(*~
		<docu>
			<summary>
				Provides switching between sequencer modes so as handling stepping tasks in th step mode.
			</summary>
		</docu>
~*)
FUNCTION_BLOCK TcoStepModeControler EXTENDS TcoState
VAR_INPUT
	inCurrentStepRunning : BOOL;
END_VAR

VAR
//	{attribute 'hide'}
	_stepBackward : TcoTask(THIS^);	
//	{attribute 'hide'}
	_stepIn : TcoTask(THIS^);	
//	{attribute 'hide'}
	_stepForward : TcoTask(THIS^);
END_VAR

THIS^._stepBackward.Enabled := THIS^.Mode = eSequencerMode.StepMode;
THIS^._stepIn.Enabled := THIS^.Mode = eSequencerMode.StepMode;
THIS^._stepForward.Enabled := THIS^.Mode = eSequencerMode.StepMode;

(*~
	<docu>
		<summary>
			Provides access to the mode of the sequencer. 
		</summary>		
	</docu>	
~*)	
PROPERTY Mode : eSequencerMode
GET
CASE SUPER^._State OF
	eSequencerMode.CyclicMode:
		Mode := eSequencerMode.CyclicMode;
	eSequencerMode.StepMode:
		Mode := eSequencerMode.StepMode;
	ELSE
		Mode := eSequencerMode.Invalid;
END_CASE
END_GET
SET
SUPER^.ChangeState(Mode);
END_SET
END_PROPERTY

METHOD PRIVATE OnStateChange
VAR_INPUT
	PreviousState	: INT;
	NewState 		: INT;
END_VAR
IF PreviousState = eSequencerMode.CyclicMode AND NewState = eSequencerMode.StepMode THEN
	_stepForward.Restore();
	_stepBackward.Restore();
	_stepIn.Restore(); 	

	IF inCurrentStepRunning THEN
		_stepIn.Enabled := TRUE;
		_stepIn.Invoke(); 	
	END_IF
END_IF

IF PreviousState = eSequencerMode.StepMode AND NewState = eSequencerMode.CyclicMode THEN
	_stepForward.Restore();
	_stepBackward.Restore();
	_stepIn.Restore(); 	
END_IF
END_METHOD

END_FUNCTION_BLOCK

(* stored: Version 1.1.0.1, ProductVersion 3.1.4024.6
   POU TcoStepModeControler: Id {bae82854-ce0e-0ab9-12e4-0141c7944f2d}, SpecialFunc None
   Property Mode: Id {8d4cb1af-ba19-0bb8-1400-30d988d71fba}
   Get Get: Id {895df049-a71d-0d24-2a10-6f8bfd7b53fa}
   Set Set: Id {de205606-d241-09de-0ee5-ac8cb916bc40}
   Method OnStateChange: Id {b7c60afe-dc93-0d5b-2752-c7f3e19a3b5e} *)
